FUNCTION_BLOCK "FB_AutoCtrl_ABCDE"
{ S7_Optimized_Access := 'TRUE' }
VERSION : 0.1
   VAR
      statExecutePulse : Bool;
      statMoveDoneOld : Bool;
      statOldStep : Int;
      statTargetPos { S7_SetPoint := 'False'} : "UDT_typePoint5";
      sRTRIGInitialPath {InstructionName := 'R_TRIG'; LibVersion := '1.0'} : R_TRIG;
      sRTRIGStart {InstructionName := 'R_TRIG'; LibVersion := '1.0'} : R_TRIG;
      sRTRIGStop {InstructionName := 'R_TRIG'; LibVersion := '1.0'} : R_TRIG;
      instMoveLinAbs {InstructionName := 'MC_MOVELINEARABSOLUTE'; LibVersion := '9.0'; S7_SetPoint := 'False'} : MC_MOVELINEARABSOLUTE;
      pts : Array[1..5] of "UDT_typePoint5";   // V8 (Phase F) blending statics — added 2026-05-17 per source spec §3.6
      statTotalDistance : LReal;   // snapshot at step-change: Euclidean(target - TCP) at start of step
      statProgress : LReal;   // 0.0 (just started) .. 1.0 (arrived) — drives early advance @ >0.5
   END_VAR

   VAR_TEMP
      tempCurrentPtIdx : Int;
      tempStepChanged : Bool;
      tempIsAutoStep : Bool;
      tempPosArray : Array[1..6] of LReal;
      tempRemaining : LReal;   // Euclidean distance from current TCP to target (this scan)
   END_VAR


BEGIN
	// =====================================================================
	// SCARA ABCDE 5-Point Continuous Auto Cycle
	// Wang Shuo / Huashili 4-REGION pattern (source spec §3.3+§3.5):
	//   REGION 1: 初始化路径 / INITIALIZE_PATH
	//   REGION 2: 启动 / START                — permissive AND → step:=10
	//   REGION 3: 停止 / STOP                 — R_TRIG → step:=0
	//   REGION 4: 自动 / AUTO main CASE       — 6 states (0/10/20/30/40/50)
	//     0=idle, 10=去A, 20=去B, 30=去C, 40=去D, 50=去E (cycle wrap 50→10)
	// ONE shared instMoveLinAbs (multi-instance) re-triggered per step on
	// rising-edge of step change. KEY to avoiding v9's OB91 overflow.
	// =====================================================================

	// =====================================================================
	// REGION 1 — INITIALIZE_PATH (source spec §2.1)
	// =====================================================================
	//

	REGION 1
	    #sRTRIGInitialPath(CLK := "GDB_MachineCmd".bo_InitPath);
	    IF #sRTRIGInitialPath.Q THEN
	        // ABCDE — square pattern in WCS, all at Z=400mm above home.
	        #pts[1].x := 1800.0;
	        #pts[1].y := 0.0;
	        #pts[1].z := 400.0;
	        #pts[1].a := 0.0;   // A
	        #pts[2].x := 1800.0;
	        #pts[2].y := 300.0;
	        #pts[2].z := 400.0;
	        #pts[2].a := 0.0;   // B
	        #pts[3].x := 1500.0;
	        #pts[3].y := 300.0;
	        #pts[3].z := 400.0;
	        #pts[3].a := 0.0;   // C
	        #pts[4].x := 1500.0;
	        #pts[4].y := -300.0;
	        #pts[4].z := 400.0;
	        #pts[4].a := 0.0;   // D
	        #pts[5].x := 1800.0;
	        #pts[5].y := -300.0;
	        #pts[5].z := 400.0;
	        #pts[5].a := 0.0;   // E
	        "GDB_MachineCmd".bo_PathInitialed := TRUE;
	    END_IF;
	END_REGION

	// =====================================================================
	// REGION 2 — START (source spec §2.2)
	// =====================================================================
	REGION 2
	#sRTRIGStart(CLK := "GDB_MachineCmd".bo_Start);
	IF "GDB_MachineCmd".bo_Mode
	    AND "GDB_MachineCmd".bo_ESTOP_LOCK
	    AND ("GDB_MachineCmd".i16_AutoStep = 0)
	    AND #sRTRIGStart.Q
	    AND "GDB_MachineCmd".bo_PathInitialed
	    AND NOT "GDB_MachineCmd".bo_Alarm
	THEN
	    "GDB_MachineCmd".i16_AutoStep := 10;
	END_IF;


	END_REGION
	// =====================================================================
	// REGION 3 — STOP (source spec §2.3)
	// =====================================================================
	REGION 3
	    #sRTRIGStop(CLK := "GDB_MachineCmd".bo_Stop);
	    IF #sRTRIGStop.Q THEN
	        "GDB_MachineCmd".i16_AutoStep := 0;
	    END_IF;

	END_REGION


	// =====================================================================
	// REGION 4 — AUTO main CASE (source spec §3.3, 6 states)
	// =====================================================================
	//
	REGION 4
	    // Detect step-change for Execute pulse
	    #tempStepChanged := ("GDB_MachineCmd".i16_AutoStep <> #statOldStep);
	    #statOldStep := "GDB_MachineCmd".i16_AutoStep;
	    // Classify current step as "active auto step" [10..50]
	    #tempIsAutoStep := ("GDB_MachineCmd".i16_AutoStep >= 10)
	    AND ("GDB_MachineCmd".i16_AutoStep <= 50);
	    // Map step → point index (10→1, 20→2, 30→3, 40→4, 50→5)
	    IF #tempIsAutoStep THEN
	        #tempCurrentPtIdx := "GDB_MachineCmd".i16_AutoStep / 10;
	        #statTargetPos := #pts[#tempCurrentPtIdx];
	    END_IF;
	    // Execute pulse: high for ONE scan when entering a new auto step
	    #statExecutePulse := #tempStepChanged AND #tempIsAutoStep;
	    // Build the 6-element Position array (4 used + 2 trailing zeros)
	    #tempPosArray[1] := #statTargetPos.x;
	    #tempPosArray[2] := #statTargetPos.y;
	    #tempPosArray[3] := #statTargetPos.z;
	    #tempPosArray[4] := #statTargetPos.a;
	    #tempPosArray[5] := 0.0;
	    #tempPosArray[6] := 0.0;
	    // Drive MC_MoveLinearAbsolute on the kinematic group.
	    // Whole-array Position passing per v9 FB_TestRawMoveLinAbs.scl line 45.
	    #instMoveLinAbs(AxesGroup := "ScaraArm3D",
	                    Execute := #statExecutePulse,
	                    Position := #tempPosArray,
	                    Velocity := 300.0,
	                    Acceleration := 3000.0,
	                    Deceleration := 3000.0,
	                    Jerk := 30000.0,
	                    BufferMode := 5);   // 5 = BM_BLENDING_HIGH (V8/Phase F, source spec §3.6). Was 1=BM_BUFFERED.

	END_REGION
	// === V8 / Phase F: progress-based advance (source spec §3.6) ===
	// Replaces the .Done-triggered advance. Each scan, compute remaining Euclidean
	// distance from current TCP to target; snapshot at step-change as statTotalDistance;
	// advance when progress > 50% (current motion half-done; next motion queues into the
	// MC_MoveLinAbs buffer via BLENDING_HIGH; SCARA blends through the corner).
	#tempRemaining := SQRT(SQR(#statTargetPos.x - "ScaraArm3D".Tcp.x)
	                    + SQR(#statTargetPos.y - "ScaraArm3D".Tcp.y)
	                    + SQR(#statTargetPos.z - "ScaraArm3D".Tcp.z));
	IF #tempStepChanged AND #tempIsAutoStep THEN
	    #statTotalDistance := #tempRemaining;
	END_IF;
	IF #statTotalDistance > 0.001 THEN
	    #statProgress := 1.0 - #tempRemaining / #statTotalDistance;
	ELSE
	    #statProgress := 0.0;
	END_IF;
	IF #statProgress > 0.5 AND #tempIsAutoStep THEN
	    IF "GDB_MachineCmd".i16_AutoStep = 50 THEN
	        "GDB_MachineCmd".i16_AutoStep := 10;        // cycle wrap E → A (§3.5)
	    ELSE
	        "GDB_MachineCmd".i16_AutoStep :=
	        "GDB_MachineCmd".i16_AutoStep + 10;     // 10→20→30→40→50
	    END_IF;
	END_IF;
	#statMoveDoneOld := #instMoveLinAbs.Done;  // kept for diagnostic visibility
END_FUNCTION_BLOCK

